FUNCTION_BLOCK Motor_Enable
VAR_INPUT
	EnableMotor:INT :=0;
	SpeedPWM:INT;
	PositiveDirection: BOOL;
	NegativeDirection: BOOL;
END_VAR
VAR_OUTPUT
	setEnable: INT;
	setSpeedPWM:INT; 
END_VAR
VAR
	move_enabled: BOOL;
END_VAR
VAR // added by the converter: edge detectors and wires of the graphical bodies
    _w1 : BOOL;
END_VAR

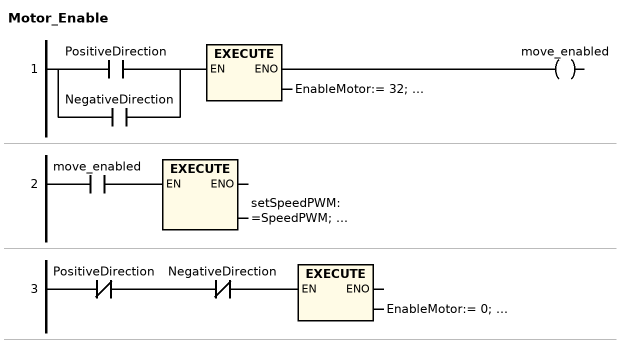
// NETWORK 1
_w1 := PositiveDirection OR NegativeDirection;
IF _w1 THEN
    EnableMotor:= 32;
    setEnable := EnableMotor;
END_IF
move_enabled := _w1;

// NETWORK 2
IF move_enabled THEN setSpeedPWM:=SpeedPWM; END_IF

// NETWORK 3
IF NOT PositiveDirection AND NOT NegativeDirection THEN
    EnableMotor:= 0;
    SpeedPWM:=0;
    setEnable := EnableMotor;
    setSpeedPWM:=SpeedPWM;
END_IF

END_FUNCTION_BLOCK

(* stored: Version 1.1.0.1, ProductVersion 3.1.4024.12
   POU Motor_Enable: Id {6b1b4b10-fbd2-4184-b8c1-f01bb9c7c68a}, SpecialFunc None *)
